TYPE Valve :
STRUCT
	extend 		 : BOOL;
	retract		 : BOOL;
	extended 	 : BOOL;
	retracted 	 : BOOL;	
END_STRUCT
END_TYPE

(* stored: Version 1.1.0.1, ProductVersion 3.1.4024.12
   DUT Valve: Id {164df541-7fba-4d4c-948b-1cbd7aa60e7d} *)
